// TIA Portal V20 program export: 0 tag tables, 0 data types, 0 data blocks, 3 code blocks (in call order from the OBs), 0 instance data blocks

ORGANIZATION_BLOCK "Main"   // OB1, LAD, ProgramCycle
TITLE = "Main Program Sweep (Cycle)"
{ S7_Optimized_Access := 'TRUE' }
// stored: SetENOAutomatically false
   VAR_INPUT
      Initial_Call : Bool;   // Initial call of this OB
      Remanence : Bool;   // =True, if remanent data are available
   END_VAR
BEGIN

REGION Network 1
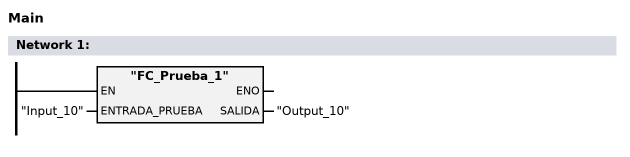
   RUNG wire#powerrail
      "FC_Prueba_1"(ENTRADA_PRUEBA := "Input_10", SALIDA => "Output_10")
   END_RUNG
   // the same network as SCL:
   "FC_Prueba_1"(ENTRADA_PRUEBA := "Input_10", SALIDA => "Output_10");
END_REGION
END_ORGANIZATION_BLOCK

FUNCTION "FC_Prueba_1" : Void   // FC1, LAD
{ S7_Optimized_Access := 'TRUE' }
// stored: SetENOAutomatically false
   VAR_INPUT
      ENTRADA_PRUEBA : Bool;
   END_VAR
   VAR_OUTPUT
      SALIDA : Bool;
   END_VAR
BEGIN

REGION Network 1
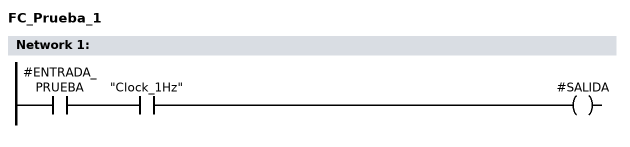
   RUNG wire#powerrail
      Contact( #ENTRADA_PRUEBA )
      Contact( "Clock_1Hz" )
      Coil( #SALIDA )
   END_RUNG
   // the same network as SCL:
   #SALIDA := #ENTRADA_PRUEBA AND "Clock_1Hz";
END_REGION
END_FUNCTION

FUNCTION "FC_Prueba_2" : Void   // FC2, LAD
{ S7_Optimized_Access := 'TRUE' }
// stored: SetENOAutomatically false
   VAR_INPUT
      ENTRADA_PRUEBA : Bool;
   END_VAR
   VAR_OUTPUT
      SALIDA : Bool;
   END_VAR
BEGIN

REGION Network 1
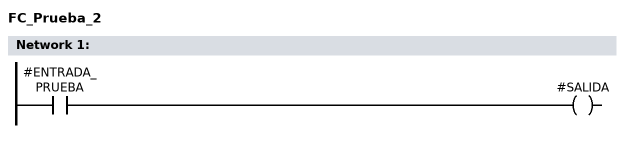
   RUNG wire#powerrail
      Contact( #ENTRADA_PRUEBA )
      Coil( #SALIDA )
   END_RUNG
   // the same network as SCL:
   #SALIDA := #ENTRADA_PRUEBA;
END_REGION
END_FUNCTION
